{attribute 'linkalways'} 
{attribute 'no_explicit_call' := 'This FB is a CLASS and must be accessed using methods or properties'}
{attribute 'enable_dynamic_creation'}
FUNCTION_BLOCK _DINT EXTENDS NumericDatatypeBase Implements I_DINT
VAR
	localData : DINT;
	activeData : REFERENCE TO DINT REF= localData;
END_VAR

PROPERTY PUBLIC Address : PVOID
GET
Address := ADR(activeData);
END_GET
END_PROPERTY

METHOD PUBLIC ClearReference
VAR_INPUT
END_VAR
activeData REF= localData;
END_METHOD

METHOD PUBLIC Clone : I_Datatype
VAR
    pClone : POINTER TO _DINT;
END_VAR
pClone := __NEW(_DINT(InitialValue := Value));
Clone := pClone^;
END_METHOD

METHOD FB_init : BOOL
VAR_INPUT
	bInitRetains : BOOL; // if TRUE, the retain variables are initialized (warm start / cold start)
	bInCopyCode : BOOL;  // if TRUE, the instance afterwards gets moved into the copy code (online change)
	InitialValue : DINT;
END_VAR
localData := InitialValue;
END_METHOD

PROPERTY PUBLIC IsEven : BOOL
GET
IsEven := (Value mod 2) = 0;
END_GET
END_PROPERTY

PROPERTY PUBLIC IsFloat : BOOL
GET
IsFloat := FALSE;
END_GET
END_PROPERTY

PROPERTY PUBLIC IsSigned : BOOL
GET
IsSigned := TRUE;
END_GET
END_PROPERTY

METHOD PUBLIC MakeReferenceTo
VAR_INPUT
	ReferenceTarget : REFERENCE TO DINT;
END_VAR
activeData REF= ReferenceTarget;
END_METHOD

PROPERTY PUBLIC MaxValue : DINT
GET
MaxValue := DatatypeLimits.DINT_MAX_VALUE;
END_GET
END_PROPERTY

PROPERTY PUBLIC MinValue : DINT
GET
MinValue := DatatypeLimits.DINT_MIN_VALUE;
END_GET
END_PROPERTY

METHOD PROTECTED SerializeMaxValue
VAR_INPUT
	Serializer : I_Serializer;
END_VAR
Serializer.AddDint(MaxValue);
END_METHOD

METHOD PROTECTED SerializeMinValue
VAR_INPUT
	Serializer : I_Serializer;
END_VAR
Serializer.AddDint(MinValue);
END_METHOD

METHOD PUBLIC SerializeWith
VAR_INPUT
	Serializer : I_Serializer;
END_VAR
Serializer.AddDint(activeData);
END_METHOD

PROPERTY PUBLIC Size : UDINT
GET
Size := SIZEOF(activeData);
END_GET
END_PROPERTY

METHOD PUBLIC TryConvertTo : BOOL
VAR_INPUT
	Destination : ANY;
END_VAR
TryConvertTo := TryConvert_DINT_To_Destination(activeData, Destination);
END_METHOD

METHOD PUBLIC TryConvertTo_ : BOOL
VAR_INPUT
	Destination : I_Datatype;
END_VAR
VAR
	resultofBitConversion : BOOL;
	destinationAs_BIT : I_BIT;
	destinationAs_BOOL : I_BOOL;
	destinationAs_BYTE : I_BYTE;
	destinationAs_DINT : I_DINT;
	destinationAs_DT : I_DT;
	destinationAs_DWORD : I_DWORD;
	destinationAs_INT : I_INT;
	destinationAs_LINT : I_LINT;
	destinationAs_LREAL : I_LREAL;
	destinationAs_LWORD : I_LWORD;
	destinationAs_REAL : I_REAL;
	destinationAs_SINT : I_SINT;
	destinationAs_STRING : I_STRING;
	destinationAs_TOD : I_TOD;
	destinationAs_UDINT : I_UDINT;
	destinationAs_UINT : I_UINT;
	destinationAs_ULINT : I_ULINT;
	destinationAs_USINT : I_USINT;
	destinationAs_WORD : I_WORD;
END_VAR
IF destination.TryResolveAs_BIT(destinationAs_BIT) AND_THEN TryConvert_DINT_TO_BOOL(activeData, resultofBitConversion) THEN
	destinationAs_BIT.Value := resultOfBitConversion;
	TryConvertTo_ := TRUE;
	RETURN;
END_IF

IF destination.TryResolveAs_BOOL(destinationAs_BOOL) THEN
	TryConvertTo_ := TryConvert_DINT_TO_BOOL(activeData, destinationAs_BOOL.Value);
	RETURN;
END_IF
		
IF destination.TryResolveAs_BYTE(destinationAs_BYTE) THEN
	TryConvertTo_ := TryConvert_DINT_TO_BYTE(activeData, destinationAs_BYTE.Value);
	RETURN;
END_IF

IF destination.TryResolveAs_DINT(destinationAs_DINT) THEN
	TryConvertTo_ := TryConvert_DINT_TO_DINT(activeData, destinationAs_DINT.Value);
	RETURN;
END_IF

IF destination.TryResolveAs_DT(destinationAs_DT) THEN
	TryConvertTo_ := TryConvert_DINT_TO_DT(activeData, destinationAs_DT.Value);
	RETURN;
END_IF

IF destination.TryResolveAs_DWORD(destinationAs_DWORD) THEN
	TryConvertTo_ := TryConvert_DINT_TO_DWORD(activeData, destinationAs_DWORD.Value);
	RETURN;
END_IF

IF destination.TryResolveAs_INT(destinationAs_INT) THEN
	TryConvertTo_ := TryConvert_DINT_TO_INT(activeData, destinationAs_INT.Value);
	RETURN;
END_IF

IF destination.TryResolveAs_LINT(destinationAs_LINT) THEN
	TryConvertTo_ := TryConvert_DINT_TO_LINT(activeData, destinationAs_LINT.Value);
	RETURN;
END_IF

IF destination.TryResolveAs_LREAL(destinationAs_LREAL) THEN
	TryConvertTo_ := TryConvert_DINT_TO_LREAL(activeData, destinationAs_LREAL.Value);
	RETURN;
END_IF

IF destination.TryResolveAs_LWORD(destinationAs_LWORD) THEN
	TryConvertTo_ := TryConvert_DINT_TO_LWORD(activeData, destinationAs_LWORD.Value);
	RETURN;
END_IF

IF destination.TryResolveAs_REAL(destinationAs_REAL) THEN
	TryConvertTo_ := TryConvert_DINT_TO_REAL(activeData, destinationAs_REAL.Value);
	RETURN;
END_IF

IF destination.TryResolveAs_SINT(destinationAs_SINT) THEN
	TryConvertTo_ := TryConvert_DINT_TO_SINT(activeData, destinationAs_SINT.Value);
	RETURN;
END_IF

IF destination.TryResolveAs_STRING(destinationAs_STRING) THEN
	TryConvertTo_ := TryConvert_DINT_TO_STRING(activeData, destinationAs_STRING.Value);
	RETURN;
END_IF

IF destination.TryResolveAs_TOD(destinationAs_TOD) THEN
	TryConvertTo_ := TryConvert_DINT_TO_TOD(activeData, destinationAs_TOD.Value);
	RETURN;
END_IF

IF destination.TryResolveAs_UDINT(destinationAs_UDINT) THEN
	TryConvertTo_ := TryConvert_DINT_TO_UDINT(activeData, destinationAs_UDINT.Value);
	RETURN;
END_IF

IF destination.TryResolveAs_UINT(destinationAs_UINT) THEN
	TryConvertTo_ := TryConvert_DINT_TO_UINT(activeData, destinationAs_UINT.Value);
	RETURN;
END_IF

IF destination.TryResolveAs_ULINT(destinationAs_ULINT) THEN
	TryConvertTo_ := TryConvert_DINT_TO_ULINT(activeData, destinationAs_ULINT.Value);
	RETURN;
END_IF

IF destination.TryResolveAs_USINT(destinationAs_USINT) THEN
	TryConvertTo_ := TryConvert_DINT_TO_USINT(activeData, destinationAs_USINT.Value);
	RETURN;
END_IF

IF destination.TryResolveAs_WORD(destinationAs_WORD) THEN
	TryConvertTo_ := TryConvert_DINT_TO_WORD(activeData, destinationAs_WORD.Value);
	RETURN;
END_IF
END_METHOD

METHOD TryDeserializeFrom : BOOL
VAR_INPUT
	Deserializer : I_Deserializer;
	Feedback : I_DeserializerFeedback;
END_VAR
TryDeserializeFrom := Deserializer.TryGetDint(activeData, Feedback);
END_METHOD

METHOD TryMakeReferenceTo : BOOL
VAR_INPUT
	Target : I_Datatype;
END_VAR
VAR
	pTargetData : POINTER TO DINT;
END_VAR
IF NOT IsEquivalentTo(Target) THEN
	RETURN;
END_IF

pTargetData := Target.Address;
activeData REF= pTargetData^;
TryMakeReferenceTo := TRUE;
END_METHOD

METHOD PUBLIC TryResolveAs_DINT : BOOL
VAR_INPUT
	Destination : REFERENCE TO I_DINT;
END_VAR
Destination := THIS^;
TryResolveAs_DINT := TRUE;
END_METHOD

PROPERTY PUBLIC TypeName : T_MAXSTRING
GET
TypeName := 'DINT';
END_GET
END_PROPERTY

{warning disable C5410}
PROPERTY PUBLIC Value : REFERENCE TO DINT
{warning restore C5410}
GET
Value REF= activeData;
END_GET
END_PROPERTY

END_FUNCTION_BLOCK

(* stored: Version 1.1.0.1, ProductVersion 3.1.4026.13
   POU _DINT: Id {90897d60-de15-4541-a8aa-871c9684610b}, SpecialFunc None
   Folder Constructor: Id {a856f573-98c4-40d1-9309-318f16e2657c}
   Folder Protected: Id {4470f3df-698e-4a92-a180-e11accbb6f57}
   Property Address: Id {8728a38b-5420-4fae-886c-e62a24ac265c}
   Get Get: Id {7b7cac06-6447-4ae3-a794-149c42497105}
   Method ClearReference: Id {7e36b9ec-a508-4109-964f-b05eed586f2a}
   Method Clone: Id {eb909221-4525-42ac-a017-259260165d4e}
   Method FB_init: Id {3cd50833-2c7f-498a-a2ce-d24c1316c2ec}
   Property IsEven: Id {867efce6-1f88-0522-2b05-61cbfc757dc4}
   Get Get: Id {f65d136f-8978-061c-1518-3cdeefb76121}
   Property IsFloat: Id {0af31b1e-5c04-4e03-9ec8-e09e65f01eb2}
   Get Get: Id {5e308476-9dc8-4be4-8231-0e96d70dcd92}
   Property IsSigned: Id {e4b5fb3f-6b52-4b0d-a341-9db5e3b1cda6}
   Get Get: Id {082ad492-75ce-4872-ab26-8c27fc203f3c}
   Method MakeReferenceTo: Id {3424f025-ae04-4c0c-8414-aae0d36b62ea}
   Property MaxValue: Id {0159c5c3-1763-4d78-bdd6-ace8b31fa1df}
   Get Get: Id {151ad154-7187-45e4-8a54-7bfb69a4c877}
   Property MinValue: Id {2dc25eb8-63ce-4a6f-bf5d-af422860e06a}
   Get Get: Id {3625e045-6e8d-43f9-ab6c-9a4780107eec}
   Method SerializeMaxValue: Id {ebbf42cf-a89b-421f-ae93-a52b5fca4620}
   Method SerializeMinValue: Id {1a38d650-ea10-473e-9a7f-8ca08f4895be}
   Method SerializeWith: Id {a15b37b9-6b28-4a5c-8555-ebc8d08318d8}
   Property Size: Id {3d0505ba-35d8-4a59-915b-c790ecc22532}
   Get Get: Id {c468404e-baef-4ab1-9002-71fa1a256bf1}
   Method TryConvertTo: Id {4d0a818a-0f9e-04e4-234e-34da6cab4a3c}
   Method TryConvertTo_: Id {1282644a-cd47-052b-2a03-7da42904d031}
   Method TryDeserializeFrom: Id {458cd8ee-b204-4a15-9f39-262426569b8f}
   Method TryMakeReferenceTo: Id {f51951c3-e009-4bad-b3bd-934e2a11edbf}
   Method TryResolveAs_DINT: Id {0655997e-2d74-084f-12ff-f84ace469804}
   Property TypeName: Id {0f65fc63-d29d-45b3-8dae-d69702c17699}
   Get Get: Id {bc4c68c9-3607-4ab0-8894-8d44e7542e0d}
   Property Value: Id {bcb8f7c5-7aaa-46ea-bcef-de9d6a0b3933}
   Get Get: Id {1d5ab7c2-66ec-4a07-bc9d-5b8f067dad9a} *)
